// TwinCAT 3 PLC project PLC
// ProgramVersion: 3.1.4026.24
// libraries:
//   Tc2_ModbusRTU, * (Beckhoff Automation GmbH)
//   Tc2_Standard, * (Beckhoff Automation GmbH)
//   Tc2_System, * (Beckhoff Automation GmbH)
//   Tc3_AnyBuffer, * (KimRo)
// project tree:
//   / BGComm.TcTTO, PlcTask.TcTTO
//   Components/ModbusDeviceSample/ ModbusDevice.TcPOU (not stored), ModbusDint.TcDUT, ModbusReal.TcDUT, ST_ModbusDevice_HMI.TcDUT (not stored), ST_ModbusDeviceParam.TcDUT
//   Components/ModbusHandler/datatypes/ E_ModbusFunction.TcDUT (not stored), ST_ModbusCommand.TcDUT (not stored)
//   Components/ModbusHandler/ I_ModbusHandler.TcIO (not stored), ModbusHandler_KL6x22B.TcPOU, ModbusHandler_KL6x5B.TcPOU (not stored), ModbusHandler_PcCOM.TcPOU
//   Program/ BG_Communication.TcPOU (not stored), MAIN.TcPOU (not stored), Param.TcGVL
// real-time tasks:
//   TASK PlcTask: cycle T#10ms, priority 8, ADS port 350
//   TASK BGComm: cycle T#1ms, priority 4, ADS port 351
//   TASK PlcTask1: cycle T#10ms, priority 20, ADS port 352
// I/O:
//   DEVICE Device 1 (EtherCAT), AmsNetId 169.254.218.108.2.1
//     Term 1 (EK1200) [EK1200-5000 EtherCAT Power supply (2A E-Bus)]
//       Term 2 (EL6022) [EL6022 Interface 2Ch. (RS422/485)]
// variable links:
//   (this object) <-> Device 1 (EtherCAT)/Term 1 (EK1200)/Term 2 (EL6022)
//     BGComm Inputs/BG_Communication.modbushandler._Terminal.InData @bit {16..184 step 8} <-> COM Inputs Channel 1/Data In {0..21}  (22 links)
//     BGComm Inputs/BG_Communication.modbushandler._Terminal.InData <-> COM Inputs Channel 1/Status
//     BGComm Inputs/BG_Communication.modbushandler._Terminal.WcState <-> WcState/WcState
//     BGComm Outputs/BG_Communication.modbushandler._Terminal.OutData <-> COM Outputs Channel 1/Ctrl
//     BGComm Outputs/BG_Communication.modbushandler._Terminal.OutData @bit {16..184 step 8} <-> COM Outputs Channel 1/Data Out {0..21}  (22 links)

CONFIGURATION PLC
    RESOURCE PLC ON TwinCAT3
        TASK BGComm(INTERVAL := T#1ms, PRIORITY := 4);
        TASK PlcTask(INTERVAL := T#10ms, PRIORITY := 8);
        PROGRAM BG_Communication WITH BGComm : BG_Communication;
        PROGRAM MAIN WITH PlcTask : MAIN;
    END_RESOURCE
END_CONFIGURATION

// ---- Components/ModbusDeviceSample/ModbusDint.TcDUT
TYPE ModbusDint :
UNION
	rawdata		: ARRAY[0..1] OF WORD;
	value	: DINT;
END_UNION
END_TYPE

// ---- Components/ModbusDeviceSample/ModbusReal.TcDUT
TYPE ModbusReal :
UNION
	rawdata		: ARRAY[0..1] OF WORD;
	value		: REAL;
END_UNION
END_TYPE

// ---- Components/ModbusDeviceSample/ST_ModbusDeviceParam.TcDUT
TYPE ST_ModbusDeviceParam :
STRUCT
	MBSAdress			: BYTE	:= 30;
	UpdateTime			: TIME	:= T#1000MS;
END_STRUCT
END_TYPE

// ---- Program/Param.TcGVL
VAR_GLOBAL CONSTANT
	MAXMODBUSBUFFER	: UINT := 200;
END_VAR

// ---- Components/ModbusHandler/ModbusHandler_KL6x22B.TcPOU
// Queue-based Modbus RTU command handler with ringbuffer
{attribute 'no_explicit_call' := 'do not call this POU directly'}
FUNCTION_BLOCK ModbusHandler_KL6x22B IMPLEMENTS I_ModbusHandler
VAR_INPUT
END_VAR
VAR_OUTPUT
END_VAR
VAR
	_Terminal							: Tc2_ModbusRTU.ModbusRtuMasterV2_KL6x22B;
END_VAR
VAR
	_Busy								: BOOL;
	_Error								: BOOL;
	_ErrorId								: MODBUS_ERRORS;
	_ModbusTimeout						: TIME := T#500MS;	
	_commandToProcess					: ST_ModbusCommand;
	_bufferHandler						: Tc3_AnyBuffer.FifoBuffer(_buffer,TRUE,FALSE);
	_buffer								: Tc3_AnyBuffer.AnyBuffer(_arBuffer,0,param.MAXMODBUSBUFFER,FALSE);
	_arBuffer							: ARRAY[0..MAXMODBUSBUFFER] OF ST_ModbusCommand;
	_bufferLock							: BOOL;
END_VAR
VAR CONSTANT
	ERROR_RESULT						: hresult := e_fail;
	OK_RESULT							: hresult := s_ok;
END_VAR

METHOD AddToBuffer : Hresult
VAR_INPUT
	command			: ST_ModbusCommand;
END_VAR
VAR CONSTANT
	PENDING_RESULT		: hresult := S_Pending;
END_VAR
// Set status to pending and add to ringbuffer
IF Tc2_System.TestAndSet(_bufferLock) THEN
	MEMCPY(destAddr:= command.Result,srcAddr:=ADR(PENDING_RESULT),n:=SIZEOF(PENDING_RESULT));
	_bufferHandler.Push(command);
	
	AddToBuffer := s_ok;
	_bufferLock:=FALSE;
ELSE
	AddToBuffer := e_fail;
END_IF
END_METHOD

PROPERTY Busy : bool
GET
Busy			:= _Busy;
END_GET
END_PROPERTY

METHOD Cyclic
(*----------------------------------------------------------------------
Wait for a new bufferd command to process
-----------------------------------------------------------------------*)
	// Check for queued commands
	IF NOT _Busy AND NOT _bufferLock THEN
		IF NOT _bufferHandler.isEmpty THEN
			_Error := FALSE;
			_ErrorId	:= 0;
			_Busy								:= _bufferHandler.Pop(_commandToProcess);
		END_IF
	END_IF
		
	(*----------------------------------------------------------------------
	Process command
	-----------------------------------------------------------------------*)
	IF _Busy AND _commandToProcess.Result <> 0 THEN
			// Copy parameters to modbus FB
			_Terminal.UnitID    		:= _commandToProcess.UnitID;
			_Terminal.Quantity  		:= _commandToProcess.Quantity;
			_Terminal.MBAddr    		:= _commandToProcess.MBAddr;
			_Terminal.cbLength		:= _commandToProcess.cbLength;
			_Terminal.Timeout			:= _ModbusTimeout;
			_Terminal.pMemoryAddr 	:= _commandToProcess.pMemoryAddr;

		CASE _commandToProcess.ModbusFunction OF
			E_ModbusFunction.ReadCoils:
				_Terminal.readcoils(	execute := TRUE,
									);
			E_ModbusFunction.ReadInputStatus:
				_Terminal.ReadInputStatus(execute := TRUE,
									);
			E_ModbusFunction.ReadRegs	:
				_Terminal.ReadRegs(execute := TRUE,
									);
			E_ModbusFunction.ReadInputRegs :
				_Terminal.ReadInputRegs(execute := TRUE,
									);
			E_ModbusFunction.WriteSingleCoil:
				_Terminal.WriteSingleCoil(execute := TRUE);
			E_ModbusFunction.WriteSingleRegister:
				_Terminal.WriteSingleRegister(execute := TRUE);
			E_ModbusFunction.WriteMultipleCoils	:
				_Terminal.WriteMultipleCoils(execute := TRUE);
			E_ModbusFunction.WriteRegs		:
				_Terminal.WriteRegs(execute := TRUE);
			E_ModbusFunction.Diagnostics		:
				_Terminal.Diagnostics(execute := TRUE);

		END_CASE
			// Wait for completion
			IF NOT _Terminal.BUSY THEN
				
				_Terminal.readcoils(	execute := FALSE,);
				_Terminal.ReadInputStatus(execute := FALSE,);
				_Terminal.ReadRegs(execute := FALSE,);
				_Terminal.ReadInputRegs(execute := FALSE,);
				_Terminal.WriteSingleCoil(execute := FALSE);
				_Terminal.WriteSingleRegister(execute := FALSE);
				_Terminal.WriteMultipleCoils(execute := FALSE);
				_Terminal.WriteRegs(execute := FALSE
				_Terminal.Diagnostics(execute := false);
				
				_Busy									:= FALSE;
				// Write result to caller's pointer
				IF NOT _Terminal.Error THEN
					MEMCPY(destAddr:= _commandToProcess.Result,srcAddr:=ADR(OK_RESULT),n:=SIZEOF(OK_RESULT));
				ELSE
					MEMCPY(destAddr:= _commandToProcess.Result,srcAddr:=ADR(ERROR_RESULT),n:=SIZEOF(ERROR_RESULT));
					//ADSLOGSTR( msgCtrlMask := ADSLOG_MSGTYPE_ERROR, msgFmtStr := 'modbus command Failed', strArg :='');
					_Error := TRUE;
					_ErrorId	:= _Terminal.ErrorId;
				END_IF
			END_IF
		ELSIF _Busy AND _commandToProcess.Result <> 0 THEN
			//ADSLOGSTR( msgCtrlMask := ADSLOG_MSGTYPE_ERROR, msgFmtStr := 'bad command receieved', strArg :='');
			_Busy		:= FALSE;
		END_IF
END_METHOD

PROPERTY Error : bool
GET
Error		:= _Error;
END_GET
END_PROPERTY

PROPERTY Errorid : MODBUS_ERRORS
GET
Errorid		:= _ErrorId;
END_GET
END_PROPERTY

PROPERTY ModbusTimeout : Time
SET
_ModbusTimeout		:=ModbusTimeout;
END_SET
END_PROPERTY

END_FUNCTION_BLOCK

// ---- Components/ModbusHandler/ModbusHandler_PcCOM.TcPOU
// Queue-based Modbus RTU command handler with ringbuffer
{attribute 'no_explicit_call' := 'do not call this POU directly'}
FUNCTION_BLOCK ModbusHandler_PcCOM implements I_ModbusHandler
VAR_INPUT
END_VAR
VAR_OUTPUT
END_VAR
VAR
	_Terminal							: Tc2_ModbusRTU.ModbusRtuMasterV2_PcCOM;
END_VAR
VAR
	_Busy								: BOOL;
	_Error								: BOOL;
	_ErrorId								: MODBUS_ERRORS;
	_ModbusTimeout						: TIME := T#500MS;	
	_commandToProcess					: ST_ModbusCommand;
	_bufferHandler						: Tc3_AnyBuffer.FifoBuffer(_buffer,TRUE,FALSE);
	_buffer								: Tc3_AnyBuffer.AnyBuffer(_arBuffer,0,param.MAXMODBUSBUFFER,FALSE);
	_arBuffer							: ARRAY[0..MAXMODBUSBUFFER] OF ST_ModbusCommand;
	_bufferLock							: BOOL;
END_VAR
VAR CONSTANT
	ERROR_RESULT						: hresult := e_fail;
	OK_RESULT							: hresult := s_ok;
END_VAR

METHOD AddToBuffer : Hresult
VAR_INPUT
	command			: ST_ModbusCommand;
END_VAR
VAR CONSTANT
	PENDING_RESULT		: hresult := S_Pending;
END_VAR
// Set status to pending and add to ringbuffer
IF Tc2_System.TestAndSet(_bufferLock) THEN
	MEMCPY(destAddr:= command.Result,srcAddr:=ADR(PENDING_RESULT),n:=SIZEOF(PENDING_RESULT));
	_bufferHandler.Push(command);
	
	AddToBuffer := s_ok;
	_bufferLock:=FALSE;
ELSE
	AddToBuffer := e_fail;
END_IF
END_METHOD

PROPERTY Busy : bool
GET
Busy			:= _Busy;
END_GET
END_PROPERTY

METHOD Cyclic
(*----------------------------------------------------------------------
Wait for a new bufferd command to process
-----------------------------------------------------------------------*)
	// Check for queued commands
	IF NOT _Busy AND NOT _bufferLock THEN
		IF NOT _bufferHandler.isEmpty THEN
			_Error := FALSE;
			_ErrorId	:= 0;
			_Busy								:= _bufferHandler.Pop(_commandToProcess);
		END_IF
	END_IF
		
	(*----------------------------------------------------------------------
	Process command
	-----------------------------------------------------------------------*)
	IF _Busy AND _commandToProcess.Result <> 0 THEN
			// Copy parameters to modbus FB
			_Terminal.UnitID    		:= _commandToProcess.UnitID;
			_Terminal.Quantity  		:= _commandToProcess.Quantity;
			_Terminal.MBAddr    		:= _commandToProcess.MBAddr;
			_Terminal.cbLength		:= _commandToProcess.cbLength;
			_Terminal.Timeout			:= _ModbusTimeout;
			_Terminal.pMemoryAddr 	:= _commandToProcess.pMemoryAddr;

		CASE _commandToProcess.ModbusFunction OF
			E_ModbusFunction.ReadCoils:
				_Terminal.readcoils(	execute := TRUE,
									);
			E_ModbusFunction.ReadInputStatus:
				_Terminal.ReadInputStatus(execute := TRUE,
									);
			E_ModbusFunction.ReadRegs	:
				_Terminal.ReadRegs(execute := TRUE,
									);
			E_ModbusFunction.ReadInputRegs :
				_Terminal.ReadInputRegs(execute := TRUE,
									);
			E_ModbusFunction.WriteSingleCoil:
				_Terminal.WriteSingleCoil(execute := TRUE);
			E_ModbusFunction.WriteSingleRegister:
				_Terminal.WriteSingleRegister(execute := TRUE);
			E_ModbusFunction.WriteMultipleCoils	:
				_Terminal.WriteMultipleCoils(execute := TRUE);
			E_ModbusFunction.WriteRegs		:
				_Terminal.WriteRegs(execute := TRUE);
			E_ModbusFunction.Diagnostics		:
				_Terminal.Diagnostics(execute := TRUE);

		END_CASE
			// Wait for completion
			IF NOT _Terminal.BUSY THEN
				
				_Terminal.readcoils(	execute := FALSE,);
				_Terminal.ReadInputStatus(execute := FALSE,);
				_Terminal.ReadRegs(execute := FALSE,);
				_Terminal.ReadInputRegs(execute := FALSE,);
				_Terminal.WriteSingleCoil(execute := FALSE);
				_Terminal.WriteSingleRegister(execute := FALSE);
				_Terminal.WriteMultipleCoils(execute := FALSE);
				_Terminal.WriteRegs(execute := FALSE
				_Terminal.Diagnostics(execute := false);
				
				_Busy									:= FALSE;
				// Write result to caller's pointer
				IF NOT _Terminal.Error THEN
					MEMCPY(destAddr:= _commandToProcess.Result,srcAddr:=ADR(OK_RESULT),n:=SIZEOF(OK_RESULT));
				ELSE
					MEMCPY(destAddr:= _commandToProcess.Result,srcAddr:=ADR(ERROR_RESULT),n:=SIZEOF(ERROR_RESULT));
					//ADSLOGSTR( msgCtrlMask := ADSLOG_MSGTYPE_ERROR, msgFmtStr := 'modbus command Failed', strArg :='');
					_Error := TRUE;
					_ErrorId	:= _Terminal.ErrorId;
				END_IF
			END_IF
		ELSIF _Busy AND _commandToProcess.Result <> 0 THEN
			//ADSLOGSTR( msgCtrlMask := ADSLOG_MSGTYPE_ERROR, msgFmtStr := 'bad command receieved', strArg :='');
			_Busy		:= FALSE;
		END_IF
END_METHOD

PROPERTY Error : bool
GET
Error		:= _Error;
END_GET
END_PROPERTY

PROPERTY Errorid : MODBUS_ERRORS
GET
Errorid		:= _ErrorId;
END_GET
END_PROPERTY

PROPERTY ModbusTimeout : Time
SET
_ModbusTimeout		:=ModbusTimeout;
END_SET
END_PROPERTY

END_FUNCTION_BLOCK
